// TIA Portal V16 export
// export: Created 2024-12-03T15:41:46.0519135Z, ExportSetting WithReadOnly, DisplayName Totally Integrated Automation Portal, DisplayVersion V16 Update 6, DisplayName TIA Portal Version Control Interface, DisplayVersion V16 Update 2, DisplayName TIA Portal Openness, DisplayVersion V16 Update 6, DisplayName TIA Portal Teamcenter Gateway, DisplayVersion V16, DisplayName SINAMICS Startdrive Advanced, DisplayVersion V16 Update 5, DisplayName SINAMICS Startdrive G130, G150, S120, S150, SINAMICS MV, S210, DisplayVersion V16 Update 5, DisplayName SINAMICS Startdrive G110M, G120, G120C, G120D, G120P, G115D, DisplayVersion V16 Update 5, DisplayName STEP 7 Professional, DisplayVersion V16 Update 6, DisplayName STEP 7 Safety, DisplayVersion V16, DisplayName WinCC Advanced / Unified PC, DisplayVersion V16 Update 6
TYPE "Parcel_Dimensions_UDT"
// stored: CreationDate 2022-02-15T10:11:23.9492638Z, InterfaceModifiedDate 2022-02-15T10:11:35.3560495Z, IsConsistent true, LibraryConformanceStatus The object is library-conformant., ModifiedDate 2022-03-12T11:05:25.9707745Z
   STRUCT
      length : Real;
      width : Real;
      heightProduct : Real;
      heightBox : Real;
      heightBoxFinal : Real;
   END_STRUCT;
END_TYPE
